// TIA Portal project "Lab02-s7" (V16)

(* hardware
DEVICE "S7-1200 station_1"  S7-1200 Station
   slot 0: "Rack_0"  S7-1200 Rack  Rack  V1.0
   slot 1: "PLC_1"  CPU 1212C DC/DC/DC  6ES7 212-1AE40-0XB0  V4.4
*)

// ===== PLC "PLC_1"  CPU 1212C DC/DC/DC =====

VAR_GLOBAL   // PLC tag table "Tabla de variables estándar"
   "Clock_Byte" AT %MB0 : Byte;
   "Clock_10Hz" AT %M0.0 : Bool;
   "Clock_5Hz" AT %M0.1 : Bool;
   "Clock_2.5Hz" AT %M0.2 : Bool;
   "Clock_2Hz" AT %M0.3 : Bool;
   "Clock_1.25Hz" AT %M0.4 : Bool;
   "Clock_1Hz" AT %M0.5 : Bool;
   "Clock_0.625Hz" AT %M0.6 : Bool;
   "Clock_0.5Hz" AT %M0.7 : Bool;
   "System_Byte" AT %MB1 : Byte;
   "FirstScan" AT %M1.0 : Bool;
   "DiagStatusUpdate" AT %M1.1 : Bool;
   "AlwaysTRUE" AT %M1.2 : Bool;
   "AlwaysFALSE" AT %M1.3 : Bool;
   "ENTRADAI0_0" AT %I0.0 : Bool;
   "MARCA2_0" AT %M2.0 : Bool;
   "MARCA2_1" AT %M2.1 : Bool;
END_VAR

DATA_BLOCK "LOGO_S7"   // DB1
{ S7_Optimized_Access := 'FALSE' }
VERSION : 0.1
   VAR
      I1 : Bool;
      I2 : Bool;
      I3 : Bool;
      I4 : Bool;
      I5 : Bool;
      I6 : Bool;
      I7 : Bool;
      I8 : Bool;
      Q1 : Bool;
      Q2 : Bool;
      Q3 : Bool;
      Q4 : Bool;
      VW2 : Int;
      VW4 : Int;
   END_VAR
BEGIN
END_DATA_BLOCK

FUNCTION "FC_Logo_S7" : Void   // FC1, FBD
{ S7_Optimized_Access := 'TRUE' }
VERSION : 0.1
   VAR_TEMP   // added for the SCL form of the ladder/FBD networks
      _w1 : Bool;
   END_VAR
BEGIN

REGION Network 1
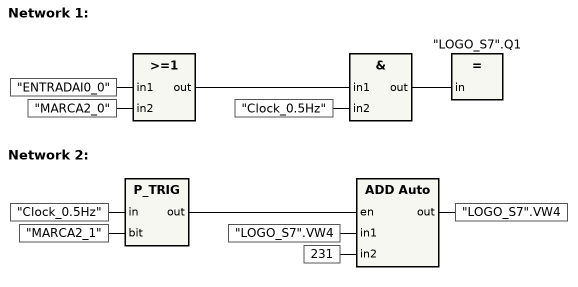
   "LOGO_S7".Q1 := ("ENTRADAI0_0" OR "MARCA2_0") AND "Clock_0.5Hz";
END_REGION

REGION Network 2
   #_w1 := "Clock_0.5Hz" AND NOT "MARCA2_1";   // rising edge
   "MARCA2_1" := "Clock_0.5Hz";
   IF #_w1 THEN "LOGO_S7".VW4 := "LOGO_S7".VW4 + 231; END_IF;
END_REGION
END_FUNCTION

ORGANIZATION_BLOCK "Main"   // OB1, LAD, ProgramCycle
TITLE = "Main Program Sweep (Cycle)"
{ S7_Optimized_Access := 'TRUE' }
VERSION : 0.1
   VAR_INPUT
      Initial_Call : Bool;   // Initial call of this OB
      Remanence : Bool;   // =True, if remanent data are available
   END_VAR
BEGIN

REGION Network 1
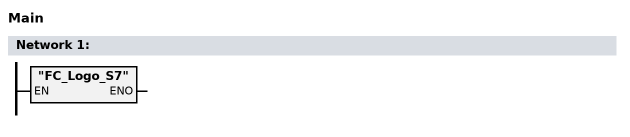
   RUNG wire#powerrail
      "FC_Logo_S7"()
   END_RUNG
   // the same network as SCL:
   "FC_Logo_S7"();
END_REGION
END_ORGANIZATION_BLOCK